(* Logix 5000 project; controller Week_4_PLC_1_Counter_UP_Counter_Down Emulate 5570 rev 30.12; software revision 30.01 *)

TASK MainTask (continuous, watchdog 500 ms) : MainProgram

MODULES
   Local : Emulate 5570 (ICP 2, rev 30.12)
END_MODULES

PROGRAM MainProgram   (* main routine MainRoutine *)
VAR
   Counter : COUNTER := (PRE := 5);
   PB1 : BOOL;
   PB2 : BOOL;
END_VAR

ROUTINE MainRoutine   (* ladder *)
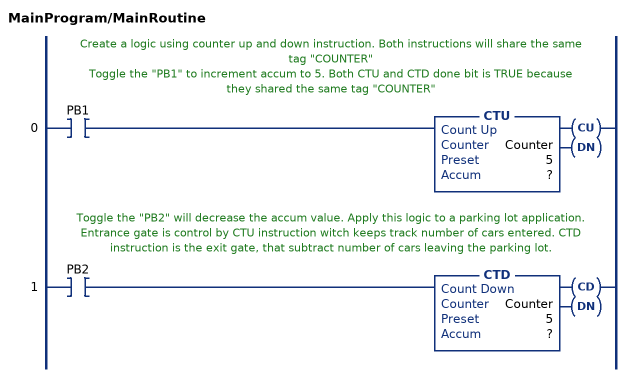
   // Create a logic using counter up and down instruction. Both instructions will share the same tag "COUNTER"
   // Toggle the "PB1" to increment accum to 5. Both CTU and CTD done bit is TRUE because they shared the same tag "COUNTER"
   0: XIC(PB1)CTU(Counter,?,?);
   // Toggle the "PB2" will decrease the accum value. Apply this logic to a parking lot application. Entrance gate is control by CTU instruction witch keeps track number of cars entered. CTD instruction is the exit gate, that subtract number of cars leaving the parking lot.
   1: XIC(PB2)CTD(Counter,?,?);
END_ROUTINE
END_PROGRAM
